// TIA Portal V20 export
DATA_BLOCK "BK06"   // DB232
// stored: MemoryReserve 100
   VAR
      "X10-1 TOP TAPE DIAMETER SENSOR" : Bool;
      "X11-1 TOP TAPE CUTTER UP" : Bool;
      "X12-1 TOP TAPE CUTTER CLAMP UP" : Bool;
      "X13-1 TOP TAPE CLAMP OPEN" : Bool;
      "X14-1 TOP TAPE TENSION BACKWARD" : Bool;
      "X15-1 TOP TAPE LOADING BACKWARD" : Bool;
      "X16-1 SPARE" : Bool;
      "X17-1 SPARE" : Bool;
      "X10-2 SPARE" : Bool;
      "X11-2 TOP TAPE CUTTER DOWN" : Bool;
      "X12-2 TOP TAPE CUTTER CLAMP DOWN" : Bool;
      "X13-2 TOP TAPE CLAMP CLOSE" : Bool;
      "X14-2 TOP TAPE TENSION FORWARD" : Bool;
      "X15-2 TOP TAPE LOADING FORWARD" : Bool;
      "X16-2 SPARE" : Bool;
      "X17-2 SPARE" : Bool;
   END_VAR
BEGIN
END_DATA_BLOCK
